RoboDK station: Final Table template.rdk

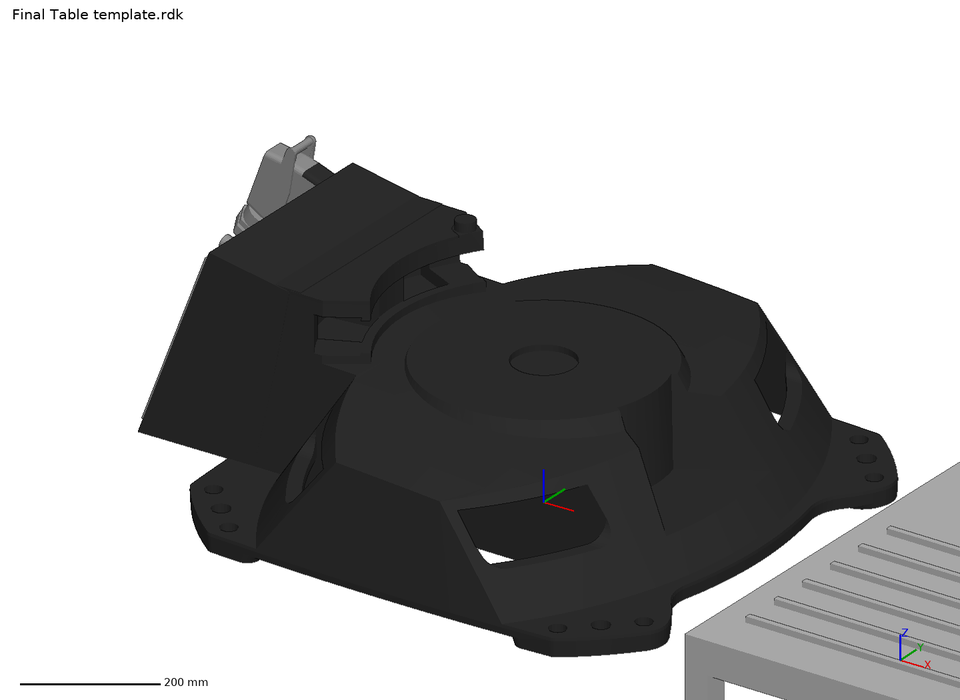
[picture v0: the station drawn from its stored meshes, robots at their saved joint values, targets as dots, program paths as lines]
Station Final Table template (saved by RoboDK 5.2.3). Poses are relative to the parent item; angles as X-Y-Z fixed-axis rotations.
  - frame KUKA KR 210 R2700 extra Base at (0, 1000, 0) mm
    - robot KUKA KR 210 R2700 extra: 6 axes, payload 210 kg, reach 2696 mm, repeatability 0.06 mm, weight 1068 kg
        joint limits [-185, -140, -120, -350, -125, -350] to [185, -5, 155, 350, 125, 350]; home [0, -90, 90, 0, 0, 0]; saved at [0, -132.562, 125.475, 0, 7.088, 0]
      - tool Spindle, TCP at (278.6, 0, 88) mm, rotated rx 0 ry 90 rz 0 deg, size 85 x 346.5 x 128 mm
  - object Table at (1700, 300, 400) mm, rotated rx 0 ry 0 rz 90 deg, size 1820 x 1605 x 465 mm
  - frame Plate 1 at (2490, 1750, 455) mm, rotated rx 0 ry 0 rz 90 deg
  - frame Plate 2 at (2490, 1310, 455) mm, rotated rx 0 ry 0 rz 90 deg
  - frame Plate 3 at (2490, 870, 455) mm, rotated rx 0 ry 0 rz 90 deg
  - frame Stringer 1 at (2490, 430, 455) mm, rotated rx 0 ry 0 rz 90 deg
  - frame Stringer 2 at (2490, 360, 455) mm, rotated rx 0 ry 0 rz 90 deg
  - frame Stringer 3 at (2490, 290, 455) mm, rotated rx 0 ry 0 rz 90 deg
  - frame Stringer 4 at (2490, 220, 455) mm, rotated rx 0 ry 0 rz 90 deg
  - frame Stringer 5 at (2490, 150, 455) mm, rotated rx 0 ry 0 rz 90 deg
  - frame Stringer 6 at (2490, 80, 455) mm, rotated rx 0 ry 0 rz 90 deg
